Fanuc KAREL source: kt00374.KL

-- PROVISIONAL review KL for V770-1; original PC SHA256 d361a708033f4e41595ac4789a2a1c66a7aa68000b3316ae3e60fbbf0a576351
-- Incomplete behavior may be omitted. Consult companion uncertainty JSON. Do not deploy.
PROGRAM KT00374
%NOLOCKGROUP
VAR
  S1 : STRING[80]
  S2 : STRING[80]
  OUT : BOOLEAN
BEGIN
  -- UNRESOLVED_PC offsets 5-14; opcodes 3F,75
  -- UNRESOLVED_PC offsets 19-28; opcodes 3F,75
  -- UNRESOLVED_PC offsets 33-42; opcodes 3F,75
  -- UNRESOLVED_PC offsets 47-56; opcodes 3F,75
  -- UNRESOLVED_PC offsets 61-80; opcodes 73,73,86,23
  -- UNRESOLVED_PC offsets 85-89; opcodes 7F
END KT00374
